// Brief: Slave Arm Run Self-check Trajectory
FUNCTION_BLOCK PUBLIC FB_SlaveCtrlSelfCheck EXTENDS FB_SlaveArmCtrlBase
VAR CONSTANT
	m_selfCheckMotionNum :INT :=1;
END_VAR
VAR
	// slave self-check motion parameters
	m_selfCheckPosture:ARRAY [1..m_selfCheckMotionNum, 1..g_sJntNum] OF LREAL:=[0.0, 	-PI/2, GVL_SlaveMotorParameters.g_maxDHJntPos[3], 	5(-g_2pi)];																			//PI/4, -PI/4, 0.3, pi, pi, pi, pi, pi];
	m_selfCheckMaxjntVel:Vec8d:=[0.2, 0.2, 0.1, 5(2.0)];
	m_selfCheckMaxjntAcc:Vec8d:=[1.0, 1.0, 0.5, 5(4.0)];
	m_selfCheckMaxjntJerk:Vec8d:=[2.0,2.0, 1.0, 5(8.0)];
	
	m_selfCheckTrajIdx: INT := 1;
	m_slefCheckPlanner: ARRAY[1..m_selfCheckMotionNum] OF FB_TrajMoveJ;
	
   // wait time for joint enable
   m_enableWaitTime :LREAL := 1.0;

   // time gap between enable and motion
   m_jntMotionTimeGap :LREAL := 0.5;

	
END_VAR

// override this function in each exact controller
METHOD PROTECTED calcCmdJntPos : BOOL
VAR_IN_OUT CONSTANT
	i_endoscopePose : ST_Frame;
	i_masterStatus :ST_MasterStatus;
	i_setupStatus: ST_SetupStatus;
	i_slaveArm :FB_SlaveArm;
END_VAR

VAR 
	i :INT;
	curJntVel :Vec8d;
END_VAR
// check if planner is ready
IF m_slefCheckPlanner[m_selfCheckTrajIdx].isGene = FALSE THEN
	calcCmdJntPos:=FALSE;
	RETURN;
END_IF

// arms enable successively
IF m_timePeriod > m_enableWaitTime THEN
       m_jntEnableFlag :=g_onesVec8i;
END_IF

IF m_timePeriod < m_enableWaitTime + m_jntMotionTimeGap THEN
	RETURN;
END_IF

// traj plan
calcCmdJntPos :=m_slefCheckPlanner[m_selfCheckTrajIdx].evaluate(m_timePeriod-m_enableWaitTime-m_jntMotionTimeGap, jntPos=> m_cmdJntPos, jntVel=>m_cmdJntVel, jntAcc=> m_cmdJntAcc);

// check if to transit to next segment
curJntVel :=i_slaveArm.curJntVel;
IF(m_timePeriod - m_enableWaitTime - m_jntMotionTimeGap > m_slefCheckPlanner[m_selfCheckTrajIdx].duration  AND norm(curJntVel)<7*GVL_SlaveControlParameters.g_jntStaticVelThres) THEN
	m_selfCheckTrajIdx:=m_selfCheckTrajIdx+1;
	m_timePeriod:=0;
END_IF

// check if to terminated
IF(m_selfCheckTrajIdx > m_selfCheckMotionNum) THEN
	m_isFinished:=TRUE;
END_IF
END_METHOD

METHOD PUBLIC init : BOOL
VAR_IN_OUT CONSTANT
	i_slaveArm	:FB_SlaveArm;
END_VAR
VAR_IN_OUT 
	r_slaveArmCtrlCmd :ST_SlaveArmCtrlCmds;
END_VAR

VAR
	i,j :INT;
	startJntPos,endJntPos :Vec8d;
	baseJntPos:Vec8d;
	cycleNum :LREAL;
END_VAR
SUPER^.Init(i_slaveArm,r_slaveArmCtrlCmd);
//m_jntEnableFlag :=g_zeroVec8i;

//set different wait time for each arm, so the arms would run self-check successively
m_enableWaitTime := i_slaveArm.armIdx-1;

// determine base joint position for instrument joint
baseJntPos :=g_zeroVec8d;
FOR i:=4 TO g_sJntNum DO
	cycleNum := FLOOR(i_slaveArm.curJntPos[i]/g_2pi);
	baseJntPos[i]:=cycleNum* g_2Pi;
END_FOR

// traj plan
// fisrt segment
// TODO: joint1/2 stay still in case arms collision
m_selfCheckTrajIdx :=1;
startJntPos:=i_slaveArm.curJntPos;
endJntPos:=startJntPos;
FOR j:=3 TO g_sJntNum DO 
	endJntPos[j]:=baseJntPos[j]+m_selfCheckPosture[1,j];
END_FOR
m_slefCheckPlanner[1].init(startJntPos,endJntPos,m_selfCheckMaxjntVel, m_selfCheckMaxjntAcc,m_selfCheckMaxjntJerk);

// other segments
IF m_selfCheckMotionNum>= 2 THEN
	FOR i:=2 TO m_selfCheckMotionNum DO 
		FOR j:=1 TO 7 DO 
			startJntPos[j]:=baseJntPos[j]+m_selfCheckPosture[i-1,j];
			endJntPos[j]:=baseJntPos[j]+m_selfCheckPosture[i,j];
		END_FOR
		m_slefCheckPlanner[i].init(startJntPos,endJntPos,m_selfCheckMaxjntVel, m_selfCheckMaxjntAcc,m_selfCheckMaxjntJerk);
	END_FOR
END_IF;

// update commands to arm
copyCmds(r_slaveArmCtrlCmd);
END_METHOD

END_FUNCTION_BLOCK

(* stored: Version 1.1.0.1, ProductVersion 3.1.4024.12
   POU FB_SlaveCtrlSelfCheck: Id {ff8ccb3f-4929-4315-b540-e9546f2dbd07}, SpecialFunc None
   Method calcCmdJntPos: Id {ffa3dbdd-63a1-4101-8d26-d1f3e6e5e2be}
   Method init: Id {c6523e12-84cb-49f8-843e-9a168bb4ce28} *)
